// Mitsubishi GX Works2 project: 42015010_0528   PLC: Q02/Q02H

PROGRAM MAIN
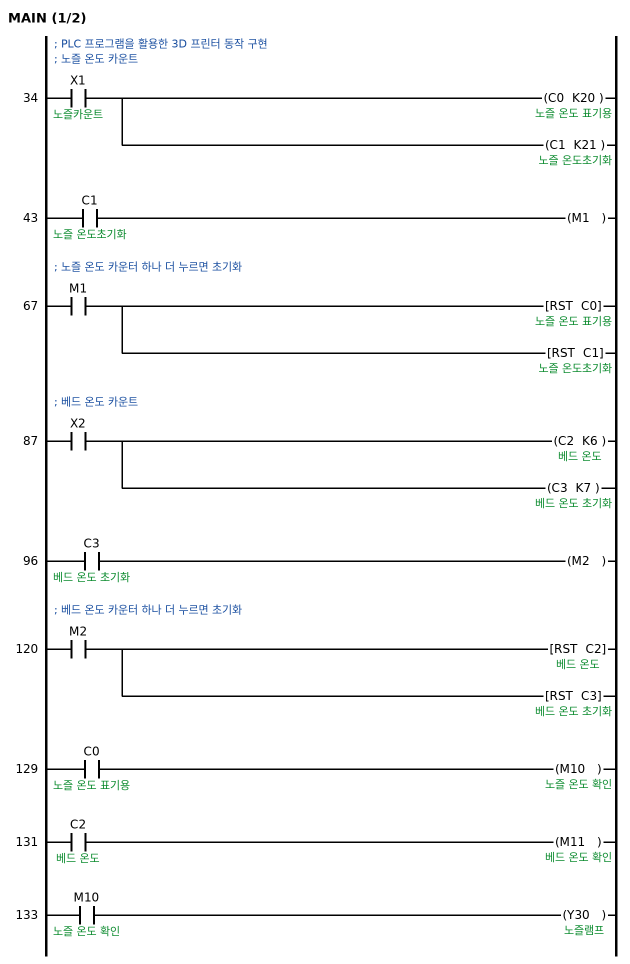
; PLC 프로그램을 활용한 3D 프린터 동작 구현
; 노즐 온도 카운트
34    LD      X1  ; 노즐카운트
      OUT     C0 K20  ; 노즐 온도 표기용
      OUT     C1 K21  ; 노즐 온도초기화
43    LD      C1  ; 노즐 온도초기화
      OUT     M1
; 노즐 온도 카운터 하나 더 누르면 초기화
67    LD      M1
      RST     C0  ; 노즐 온도 표기용
      RST     C1  ; 노즐 온도초기화
; 베드 온도 카운트
87    LD      X2
      OUT     C2 K6  ; 베드 온도
      OUT     C3 K7  ; 베드 온도 초기화
96    LD      C3  ; 베드 온도 초기화
      OUT     M2
; 베드 온도 카운터 하나 더 누르면 초기화
120   LD      M2
      RST     C2  ; 베드 온도
      RST     C3  ; 베드 온도 초기화
129   LD      C0  ; 노즐 온도 표기용
      OUT     M10  ; 노즐 온도 확인
131   LD      C2  ; 베드 온도
      OUT     M11  ; 베드 온도 확인
133   LD      M10  ; 노즐 온도 확인
      OUT     Y30  ; 노즐램프
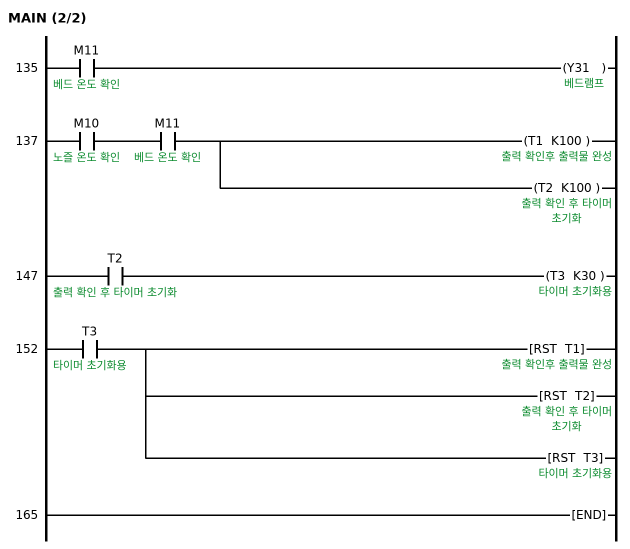
135   LD      M11  ; 베드 온도 확인
      OUT     Y31  ; 베드램프
137   LD      M10  ; 노즐 온도 확인
      AND     M11  ; 베드 온도 확인
      OUT     T1 K100  ; 출력 확인후 출력물 완성
      OUT     T2 K100  ; 출력 확인 후 타이머 초기화
147   LD      T2  ; 출력 확인 후 타이머 초기화
      OUT     T3 K30  ; 타이머 초기화용
152   LD      T3  ; 타이머 초기화용
      RST     T1  ; 출력 확인후 출력물 완성
      RST     T2  ; 출력 확인 후 타이머 초기화
      RST     T3  ; 타이머 초기화용
165   END
END_PROGRAM
